Fanuc KAREL source: WeldLWeave.kl

PROGRAM WELDLWEAVE
%NOLOCKGROUP
%NOPAUSE = ERROR + COMMAND + TPENABLE
%COMMENT = 'L weave placeholder'

BEGIN
  WRITE('WELDLWEAVE START', CR)
  WRITE('Implement L-weave motion here.', CR)
END WELDLWEAVE
